FUNCTION FC_WithinMinMax : BOOL		// Checks if the specified value is within the target range, returns TRUE if within range, FALSE otherwise
VAR_INPUT
	iValue:			LREAL;		// Value to be checked
	iMin:			LREAL;		// Target value
	iMax:			LREAL;		// This value is allowed below and above
END_VAR

FC_WithinMinMax := (iValue >= iMin) AND (iValue <= iMax);

END_FUNCTION

(* stored: Version 1.1.0.1, ProductVersion 3.1.4026.18
   POU FC_WithinMinMax: Id {2d3dbab0-dd04-443d-a193-1fb68ddf83f4}, SpecialFunc None *)
